PROGRAM MAIN
VAR
END_VAR

InterfaceTesting();
DynamicMemoryTesting();

END_PROGRAM

(* stored: Version 1.1.0.1, ProductVersion 3.1.4024.11
   POU MAIN: Id {cc66a798-1298-40f9-b59c-a64afc278fff}, SpecialFunc None *)
